(* CODESYS project CtaAppSntp_1.0.0.0.library
   Description: SNTP Library der CTA
   Version: 1.0.0.0
   Title: CtaAppSntp
   Author: SIS
   LanguageModelAttribute: qualified-access-only
   DocFormat: reStructuredText
   Placeholder: CtaAppSntp
   DefaultNamespace: CtaAppSntp
   CompiledLibraryCompatibilityVersion: CODESYS V3.5 SP16 Patch 3
   Company: CTA

Project tree, tasks and I/O mapping:
  libraries: Net Base Services, 3.5.19.20 (3S - Smart Software Solutions GmbH); CtaSysEvent, 1.0.0.0 (CTA); CtaAppTime, 1.0.0.0 (CTA)
  40 Visualizations/
  30 Program Organization Units/
    function block fbSNTP [ST]: actOnError, actSntpServer, actPeer, actUdpSend, actUdpRecive, FB_INIT, proDenyStop, proIsRegistred, metStartDone, metPrepeareStop, metCyclicCall
  00000000-0000-0000-0000-000000000000|D:\CoDeSys\LibrariesV3\trunk\Intern\CAA\CAA Template\3.4.0.0 draft\Placeholder.xml
  00000000-0000-0000-0000-000000000000|D:\CoDeSys\LibrariesV3\trunk\Intern\CAA\CAA Template\3.2.0.3 draft\Prefix.pdf
  00000000-0000-0000-0000-000000000000|D:\CoDeSys\LibrariesV3\trunk\Intern\CAA\CAA Template\3.5.2.0 draft\Placeholder.xml
  20 Structs/
  50 Images/
  10 Documenation/
    global variables VersionHistory
    global variables readMe
  21 Interface/
  11 Library Parameter/
    global variables Parameter
  12 Konstanten/
  60 Textlisten/
  13 Globale Variablen/
    global variables GVL_SNTP
*)

// 10 Documenation/VersionHistory
(* 

.. image:: ../../Images/CTA_Logo.jpg
   :align: right
   :width: 15% 

**Vorlage**   


============ =========== =========== ============================================
**Date**     **Version** **Author**  **Change**
------------ ----------- ----------- --------------------------------------------
04.03.2021   0.0.0.0     SIS         Vorlage erstellt

============ =========== =========== ============================================


*)
VAR_GLOBAL
    stInfo : STRING:= '0.0.0.0, Vorlage, CTA';
END_VAR

// 10 Documenation/readMe
(*

**ReadMe**
 
|	**Empfehlung**
|
|	Dokumentrieren Sie die Library für eine nachhaltige Entwicklung
|     
| *Beispiel* 
|
| Dies ist die Vorlage Library der CTA. Erstellen Sie ihre Library anhand dieser Vorlage.
*)

VAR_GLOBAL
    xReadMeDone              :   BOOL;
END_VAR

// 11 Library Parameter/Parameter
{attribute 'qualified_only'}
VAR_GLOBAL CONSTANT
    sIpAddr             :   NBS.IPADDRESS       := '0.0.0.0';           // IP Adresse des SNTP Server => 0.0.0.0 Erreichbar über X1 und X2       
END_VAR

// 13 Globale Variablen/GVL_SNTP
{attribute 'qualified_only'}
{attribute 'linkalways'}
VAR_GLOBAL
    fbSNTP  :   fbSNTP;  
END_VAR

// 30 Program Organization Units/fbSNTP
{attribute 'no_assign'}
FUNCTION_BLOCK fbSNTP IMPLEMENTS CtaSysEvent.ITF_APPEVENT
VAR_OUTPUT
    xError              :   BOOL;
END_VAR
VAR
    (* UDP FBs *)
    fbUdpPeer           :   NBS.UDP_Peer;
    fbUdpRecive         :   NBS.UDP_Receive; 
    fbUdpSend           :   NBS.UDP_Send;

    (* IP Fbs*)
    sIpAddr             :   NBS.IPADDRESS       := '0.0.0.0'; 
    fbIpAddr            :   NBS.IPv4Address;
    
    (* UDP Packete *)
    aybSntpSend         : ARRAY[0..67] OF BYTE;
    aybSntpRecive       : ARRAY[0..67] OF BYTE;    
    
    (* Time *)
    dtUtcDateAndTime    :   DATE_AND_TIME;    
    lwTimeStampUnix     :   LWORD;
    
    (* FOR *)
    iFor1               :   INT; 
    
    (* APP Event *)
    xIsRegistred        :   BOOL;
END_VAR

(*======================================================= SNTP(NTP) Datenstruktur =======================================================================
             
                                              0               1               2               3
                                              0 1 2 3 4 5 6 7 0 1 2 3 4 5 6 7 0 1 2 3 4 5 6 7 0 1 2 3 4 5 6 7
                                             +---+-----+-----+---------------+---------------+---------------+
                                Byte: 00-03  |LI | VN  |Mode |    Stratum    |     Poll      |   Precision   |
                                             +---------------------------------------------------------------+
                                Byte: 04-07  |  Root  Delay                                 (32 Bit)         |
                                             +---------------------------------------------------------------+
                                Byte: 08-11  |  Root  Dispersion                            (32 Bit)         |
                                             +---------------------------------------------------------------+
                                Byte: 12-15  |  Reference Identifier                        (32 Bit)         |
                                             +---------------------------------------------------------------+
                                Byte: 16-23  |  Reference Timestamp                         (64 Bit)         |
                                             |                                                               |
                                             +---------------------------------------------------------------+
                                Byte: 24-31  |  Originate Timestamp                         (64 Bit)         |
                                             |                                                               |
                                             +---------------------------------------------------------------+
                                Byte: 32-39  |  Receive Timestamp                           (64 Bit)         |
                                             |                                                               |
                                             +---------------------------------------------------------------+
                                Byte: 40-47  |  Transmit Timestamp                          (64 Bit)         |
                                             |                                                               |
                                             +---------------------------------------------------------------+
                                Byte: 48-51  |  Key Identifier      (optional)              (32 Bit)         |
                                             +---------------------------------------------------------------+
                                Byte: 52-67  |  Message Digest      (optional)              (128 Bit)        |
                                             +---------------------------------------------------------------+

=========================================================================================================================================================*)
actPeer();
actUdpRecive();
actSntpServer();
actUdpSend();
actOnError();

ACTION actOnError:
xError := fbUdpPeer.xError OR fbUdpRecive.xError OR fbUdpSend.xError OR NOT xIsRegistred;
END_ACTION

ACTION actSntpServer:
(*======================================================= SNTP(NTP) Daten aufbereitung ===================================================================
            
=========================================================================================================================================================*)
(* Leap Indicator = Flag: NO WARNING = 0 *)
aybSntpSend[0].0 := 0;  
aybSntpSend[0].1 := 0;  
(* Version Number = Flag: NTP VERSION 4 = 3 *)
aybSntpSend[0].2 := 1;  
aybSntpSend[0].3 := 1;  
aybSntpSend[0].4 := 0;  
(* Mode = Flag: SERVER = 4*)
aybSntpSend[0].5 := 0;  
aybSntpSend[0].6 := 0;  
aybSntpSend[0].7 := 1;  
(* Stratum Level = Stratum: 1 *)
aybSntpSend[1] := 1;               
(* Peer Polling Intervall 2 hoch 3 = 8 sek. *)
aybSntpSend[2] := 3;                
(* Peer Clock Precision: -6 = 134*)
aybSntpSend[3] := 134;               
(* Reference ID *)
aybSntpSend[12]:= 76;               (* L *)
aybSntpSend[13]:= 79;               (* O *)
aybSntpSend[14]:= 67;               (* C *)
aybSntpSend[15]:= 76;               (* L *)

(* Umrechnung SNTP Timestamp Base 1900-01-01 = Unix 1970-01-01 + 2208988800 sekunden *)
dtUtcDateAndTime    := CtaAppTime.FuGetDateAndTime();
lwTimeStampUnix     := DT_TO_LWORD(dtUtcDateAndTime) + LWORD#2208988800;

(* Reference Timestamp *)
aybSntpSend[16].0   := lwTimeStampUnix.24; (* Timestamp Byte 7 *)
aybSntpSend[16].1   := lwTimeStampUnix.25; (* Timestamp Byte 7 *)
aybSntpSend[16].2   := lwTimeStampUnix.26; (* Timestamp Byte 7 *)
aybSntpSend[16].3   := lwTimeStampUnix.27; (* Timestamp Byte 7 *)
aybSntpSend[16].4   := lwTimeStampUnix.28; (* Timestamp Byte 7 *)
aybSntpSend[16].5   := lwTimeStampUnix.29; (* Timestamp Byte 7 *)
aybSntpSend[16].6   := lwTimeStampUnix.30; (* Timestamp Byte 7 *)
aybSntpSend[16].7   := lwTimeStampUnix.31; (* Timestamp Byte 7 *)
                                         
aybSntpSend[17].0   := lwTimeStampUnix.16; (* Timestamp Byte 6 *)
aybSntpSend[17].1   := lwTimeStampUnix.17; (* Timestamp Byte 6 *)
aybSntpSend[17].2   := lwTimeStampUnix.18; (* Timestamp Byte 6 *)
aybSntpSend[17].3   := lwTimeStampUnix.19; (* Timestamp Byte 6 *)
aybSntpSend[17].4   := lwTimeStampUnix.20; (* Timestamp Byte 6 *)
aybSntpSend[17].5   := lwTimeStampUnix.21; (* Timestamp Byte 6 *)
aybSntpSend[17].6   := lwTimeStampUnix.22; (* Timestamp Byte 6 *)
aybSntpSend[17].7   := lwTimeStampUnix.23; (* Timestamp Byte 6 *)
                                         
aybSntpSend[18].0   := lwTimeStampUnix.08; (* Timestamp Byte 5 *)
aybSntpSend[18].1   := lwTimeStampUnix.09; (* Timestamp Byte 5 *)
aybSntpSend[18].2   := lwTimeStampUnix.10; (* Timestamp Byte 5 *)
aybSntpSend[18].3   := lwTimeStampUnix.11; (* Timestamp Byte 5 *)
aybSntpSend[18].4   := lwTimeStampUnix.12; (* Timestamp Byte 5 *)
aybSntpSend[18].5   := lwTimeStampUnix.13; (* Timestamp Byte 5 *)
aybSntpSend[18].6   := lwTimeStampUnix.14; (* Timestamp Byte 5 *)
aybSntpSend[18].7   := lwTimeStampUnix.15; (* Timestamp Byte 5 *)
                                         
aybSntpSend[19].0   := lwTimeStampUnix.00; (* Timestamp Byte 4 *)
aybSntpSend[19].1   := lwTimeStampUnix.01; (* Timestamp Byte 4 *)
aybSntpSend[19].2   := lwTimeStampUnix.02; (* Timestamp Byte 4 *)
aybSntpSend[19].3   := lwTimeStampUnix.03; (* Timestamp Byte 4 *)
aybSntpSend[19].4   := lwTimeStampUnix.04; (* Timestamp Byte 4 *)
aybSntpSend[19].5   := lwTimeStampUnix.05; (* Timestamp Byte 4 *)
aybSntpSend[19].6   := lwTimeStampUnix.06; (* Timestamp Byte 4 *)
aybSntpSend[19].7   := lwTimeStampUnix.07; (* Timestamp Byte 4 *)

aybSntpSend[20].0   := lwTimeStampUnix.56; (* Timestamp Byte 3 *)
aybSntpSend[20].1   := lwTimeStampUnix.57; (* Timestamp Byte 3 *)
aybSntpSend[20].2   := lwTimeStampUnix.58; (* Timestamp Byte 3 *)
aybSntpSend[20].3   := lwTimeStampUnix.59; (* Timestamp Byte 3 *)
aybSntpSend[20].4   := lwTimeStampUnix.60; (* Timestamp Byte 3 *)
aybSntpSend[20].5   := lwTimeStampUnix.61; (* Timestamp Byte 3 *)
aybSntpSend[20].6   := lwTimeStampUnix.62; (* Timestamp Byte 3 *)
aybSntpSend[20].7   := lwTimeStampUnix.63; (* Timestamp Byte 3 *)
                                         
aybSntpSend[21].0   := lwTimeStampUnix.48; (* Timestamp Byte 2 *)
aybSntpSend[21].1   := lwTimeStampUnix.49; (* Timestamp Byte 2 *)
aybSntpSend[21].2   := lwTimeStampUnix.50; (* Timestamp Byte 2 *)
aybSntpSend[21].3   := lwTimeStampUnix.51; (* Timestamp Byte 2 *)
aybSntpSend[21].4   := lwTimeStampUnix.52; (* Timestamp Byte 2 *)
aybSntpSend[21].5   := lwTimeStampUnix.53; (* Timestamp Byte 2 *)
aybSntpSend[21].6   := lwTimeStampUnix.54; (* Timestamp Byte 2 *)
aybSntpSend[21].7   := lwTimeStampUnix.55; (* Timestamp Byte 2 *)
                                         
aybSntpSend[22].0   := lwTimeStampUnix.40; (* Timestamp Byte 1 *)
aybSntpSend[22].1   := lwTimeStampUnix.41; (* Timestamp Byte 1 *)
aybSntpSend[22].2   := lwTimeStampUnix.42; (* Timestamp Byte 1 *)
aybSntpSend[22].3   := lwTimeStampUnix.43; (* Timestamp Byte 1 *)
aybSntpSend[22].4   := lwTimeStampUnix.44; (* Timestamp Byte 1 *)
aybSntpSend[22].5   := lwTimeStampUnix.45; (* Timestamp Byte 1 *)
aybSntpSend[22].6   := lwTimeStampUnix.46; (* Timestamp Byte 1 *)
aybSntpSend[22].7   := lwTimeStampUnix.47; (* Timestamp Byte 1 *)
                                         
aybSntpSend[23].0   := lwTimeStampUnix.32; (* Timestamp Byte 0 *)
aybSntpSend[23].1   := lwTimeStampUnix.33; (* Timestamp Byte 0 *)
aybSntpSend[23].2   := lwTimeStampUnix.34; (* Timestamp Byte 0 *)
aybSntpSend[23].3   := lwTimeStampUnix.35; (* Timestamp Byte 0 *)
aybSntpSend[23].4   := lwTimeStampUnix.36; (* Timestamp Byte 0 *)
aybSntpSend[23].5   := lwTimeStampUnix.37; (* Timestamp Byte 0 *)
aybSntpSend[23].6   := lwTimeStampUnix.38; (* Timestamp Byte 0 *)
aybSntpSend[23].7   := lwTimeStampUnix.39; (* Timestamp Byte 0 *)

(* Receive   Timestamp *)
aybSntpSend[32]     := aybSntpSend[16];     
aybSntpSend[33]     := aybSntpSend[17];
aybSntpSend[34]     := aybSntpSend[18];
aybSntpSend[35]     := aybSntpSend[19];
aybSntpSend[36]     := aybSntpSend[20];
aybSntpSend[37]     := aybSntpSend[21];
aybSntpSend[38]     := aybSntpSend[22];
aybSntpSend[39]     := aybSntpSend[23];
(* Transmit  Timestamp *)
aybSntpSend[40]     := aybSntpSend[16];
aybSntpSend[41]     := aybSntpSend[17];
aybSntpSend[42]     := aybSntpSend[18];
aybSntpSend[43]     := aybSntpSend[19];
aybSntpSend[44]     := aybSntpSend[20];
aybSntpSend[45]     := aybSntpSend[21];
aybSntpSend[46]     := aybSntpSend[22];
aybSntpSend[47]     := aybSntpSend[23];

(* Byte 0-7 von Transmit-Time auf Originate-Time umkopieren *)
FOR iFor1 := 24 TO 31 DO
    aybSntpSend[iFor1] := aybSntpRecive[iFor1 + 16];
END_FOR;
END_ACTION

ACTION actPeer:
(* IP Adr *)
sIpAddr := Parameter.sIpAddr;
fbIpAddr.SetInitialValue(ipAddress := sIpAddr);    

(* Socket Peer *)
fbUdpPeer(  xEnable         := NOT fbUdpPeer.xError,
            itfIPAddress    := fbIpAddr,
            uiPort          := 123);
END_ACTION

ACTION actUdpSend:
(* Send SNTP *)
fbUdpSend(  xExecute        := fbUdpPeer.xBusy AND NOT fbUdpSend.xDone AND fbUdpRecive.xReady AND NOT fbUdpSend.xError,
            itfPeer         := fbUdpPeer,
            itfIPAddress    := fbUdpRecive.itfIPAddressFrom,
            uiPort          := fbUdpRecive.uiPortFrom, 
            pData           := ADR(aybSntpSend),
            udiSize         := 48);
END_ACTION

ACTION actUdpRecive:
(* UDP Reccive *)
fbUdpRecive(    xEnable := fbUdpPeer.xBusy AND NOT fbUdpRecive.xReady AND NOT fbUdpRecive.xError,
                itfPeer := fbUdpPeer, 
                pData   := ADR(aybSntpRecive), 
                udiSize := 68);
END_ACTION

//FB_Init ist immer implizit verfügbar und wird primär für die Initialisierung verwendet.
//Der Rückgabewert wird nicht ausgewertet. Für gezielte Einflussnahme können Sie
//die Methoden explizit deklarieren und darin mit dem Standard-Initialisierungscode 
//zusätzlichen Code bereitstellen. Sie können den Rückgabewert auswerten.
METHOD FB_Init: BOOL
VAR_INPUT    
bInitRetains: BOOL; // TRUE: Die Retain-Variablen werden initialisiert (Reset warm / Reset kalt)    
bInCopyCode: BOOL;  // TRUE: Die Instanz wird danach in den Kopiercode kopiert (Online-Change)
END_VAR
CtaSysEvent.fcRegistry(THIS^);
END_METHOD

PROPERTY proDenyStop : BOOL
GET
proDenyStop := FALSE;
END_GET
END_PROPERTY

PROPERTY proIsRegistred : BOOL
SET
xIsRegistred := proIsRegistred;
END_SET
GET
proIsRegistred := xIsRegistred;
END_GET
END_PROPERTY

METHOD metStartDone : BOOL
RETURN;
END_METHOD

METHOD metPrepeareStop : BOOL
RETURN;
END_METHOD

METHOD metCyclicCall : BOOL
(* Self Call *)
THIS^();
END_METHOD

END_FUNCTION_BLOCK
